// TwinCAT 3 PLC project TcpServerPlc
// ProgramVersion: 3.1.4020.1
// libraries:
//   Tc2_Standard, * (Beckhoff Automation GmbH)
//   Tc2_System, * (Beckhoff Automation GmbH)
//   Tc3_Module, * (Beckhoff Automation GmbH)
// project tree:
//   DUTs/ IpAdrUnion.TcDUT
//   / PlcTask.TcTTO
//   POUs/ MAIN.TcPOU, TcpServer.TcPOU
// real-time tasks:
//   TASK PlcTask: cycle T#10ms, priority 20, ADS port 350
// I/O:
//   DEVICE Device 1 (RT-Ethernet Adapter)

CONFIGURATION TcpServerPlc
    RESOURCE PLC ON TwinCAT3
        TASK PlcTask(INTERVAL := T#10ms, PRIORITY := 20);
        PROGRAM MAIN WITH PlcTask : MAIN;
    END_RESOURCE
END_CONFIGURATION

// ---- DUTs/IpAdrUnion.TcDUT
TYPE IpAdrUnion :
UNION
	ipadrIPStack : UDINT;
	ipadr : ARRAY[0..3] OF BYTE;
END_UNION
END_TYPE

// ---- POUs/MAIN.TcPOU
PROGRAM MAIN
VAR
	tcpServer : TcpServer; 
END_VAR

tcpServer();

END_PROGRAM

// ---- POUs/TcpServer.TcPOU
{attribute 'c++_compatible'}
FUNCTION_BLOCK TcpServer IMPLEMENTS ITcIoTcpProtocolRecv
VAR_INPUT
END_VAR
VAR_OUTPUT
END_VAR
VAR
    {attribute 'TcInitSymbol'}
	oid: OTCID; 
    ipTcp:       ITcIoTcpProtocol;
    tcpPort:    UINT := 11000;
    nReceivedPakets: UINT;	
	socketId : UDINT;
	nConnectionSocket : UDINT;
	lastTcpEvent	: TCPIP_EVENT;
	lastIpAdr : IpAdrUnion;
END_VAR

IF ipTcp <> 0 THEN
    ipTcp.CheckReceived();
END_IF

METHOD FB_exit : BOOL
VAR_INPUT
	bInCopyCode : BOOL; // if TRUE, the exit method is called for exiting an instance that is copied afterwards (online change).
END_VAR
IF ipTcp <> 0 AND NOT bInCopyCode THEN // no online change
	IF (socketId <> 0) THEN  
	    ipTcp.FreeSocket(socketId);
	END_IF
	IF (nConnectionSocket <> 0) THEN  
		ipTcp.FreeSocket(nConnectionSocket);
	END_IF
	FW_SafeRelease(ADR(ipTcp));
END_IF
END_METHOD

METHOD FB_init : BOOL
VAR_INPUT
	bInitRetains : BOOL; // if TRUE, the retain variables are initialized (warm start / cold start)
	bInCopyCode : BOOL;  // if TRUE, the instance afterwards gets moved into the copy code (online change)
END_VAR
VAR
	ipSrv: ITComObjectServer;
	hr : HRESULT;
END_VAR
IF NOT bInCopyCode THEN // no online change
	IF ipTcp = 0 THEN
		hr := FW_ObjMgr_GetObjectInstance(	oid:=oid, 
												iid:=TC_GLOBAL_IID_LIST.IID_ITcIoTcpProtocol, 
												pipUnk:=ADR(ipTcp) );
		IF SUCCEEDED(hr) AND ipTcp.AllocSocket(THIS^, socketId) = 0 THEN //startup -> open port 
			IF (ipTcp.Listen(socketId, tcpPort) = 0) THEN
            	FB_init := TRUE;
			END_IF
		ELSE 
          	FB_init := FALSE;
          	FW_SafeRelease(ADR(ipTcp));
		END_IF
	END_IF
END_IF
END_METHOD

METHOD FB_reinit : BOOL
VAR_INPUT
END_VAR
IF (ipTcp <> 0 AND socketId <> 0) THEN 			//reregister THIS^ for online changes  
	ipTcp.AllocSocket(THIS^, socketId);
END_IF
IF (ipTcp <> 0 AND nConnectionSocket <> 0) THEN //reregister THIS^ for online changes  
	ipTcp.AllocSocket(THIS^, nConnectionSocket);
END_IF
END_METHOD

{attribute 'object_name' := 'ReceiveData'}
{attribute 'c++_compatible'}
{attribute 'signature_flag' := '33554688'}
{attribute 'pack_mode' := '4'}
{attribute 'show'}
{attribute 'minimal_input_size' := '4'}
{attribute 'checksuperglobal'}
METHOD ReceiveData : HRESULT
VAR_INPUT
	socketId	: UDINT;
	nData	: UDINT;
	pData	: PVOID;
END_VAR
VAR 
	sentBytes :UDINT; 
END_VAR
nReceivedPakets := nReceivedPakets+1;
IF ipTcp <> 0 THEN
	ipTcp.GetRemoteIpAddr(socketId, lastIpAdr.ipadrIPStack );
    ipTcp.SendData(socketId, nData, pData, sentBytes); // send data back
END_IF
END_METHOD

{attribute 'object_name' := 'ReceiveEvent'}
{attribute 'c++_compatible'}
{attribute 'signature_flag' := '33554688'}
{attribute 'pack_mode' := '4'}
{attribute 'show'}
{attribute 'minimal_input_size' := '4'}
{attribute 'checksuperglobal'}
METHOD ReceiveEvent : HRESULT
VAR_INPUT
	socketId	: UDINT;
	tcpEvent	: TCPIP_EVENT;
END_VAR
CASE tcpEvent OF
	TCPIP_EVENT_ERROR:
	TCPIP_EVENT_RESET:
		ipTcp.FreeSocket(socketId);
	TCPIP_EVENT_TIMEOUT:
		ipTcp.FreeSocket(socketId);
	TCPIP_EVENT_CONN_CLOSED:
		ipTcp.FreeSocket(socketId);
	TCPIP_EVENT_CONN_INCOMING:
		ipTcp.Accept(socketId);
		nConnectionSocket := socketId; //store socketid; used at least in init during onlinechange
	TCPIP_EVENT_KEEP_ALIVE:
	TCPIP_EVENT_CONN_IDLE:
	TCPIP_EVENT_DATA_SENT:
	TCPIP_EVENT_DATA_RECEIVED:
	TCPIP_EVENT_LINKCONNECT:
	TCPIP_EVENT_LINKDISCONNECT:
		ipTcp.FreeSocket(socketId);
END_CASE; 
lastTcpEvent := tcpEvent;
ReceiveEvent := S_OK;
END_METHOD

{attribute 'object_name' := 'TcAddRef'}
{attribute 'c++_compatible'}
{attribute 'signature_flag' := '33554688'}
{attribute 'pack_mode' := '4'}
{attribute 'show'}
{attribute 'minimal_input_size' := '4'}
{attribute 'checksuperglobal'}
METHOD TcAddRef : UDINT
END_METHOD

{attribute 'object_name' := 'TcQueryInterface'}
{attribute 'c++_compatible'}
{attribute 'signature_flag' := '33554688'}
{attribute 'pack_mode' := '4'}
{attribute 'show'}
{attribute 'minimal_input_size' := '4'}
{attribute 'checksuperglobal'}
METHOD TcQueryInterface : HRESULT
VAR_INPUT
	iid	: REFERENCE TO IID;
	pipItf	: POINTER TO PVOID;
END_VAR
END_METHOD

{attribute 'object_name' := 'TcRelease'}
{attribute 'c++_compatible'}
{attribute 'signature_flag' := '33554688'}
{attribute 'pack_mode' := '4'}
{attribute 'show'}
{attribute 'minimal_input_size' := '4'}
{attribute 'checksuperglobal'}
METHOD TcRelease : UDINT
END_METHOD

END_FUNCTION_BLOCK
